FUNCTION ifExprFunc2: DINT
VAR_INPUT
    state: STATE;
END_VAR


        IF (state.dvar_M_p_vf) THEN
    ifExprFunc2 := 8;
ELSE
    ifExprFunc2 := 9;
END_IF;

END_FUNCTION

(* stored: ProductVersion 3.1.0.18, Version 1.1.0.1 *)
